# EPICS StreamDevice protocol: pt2025Sup/pt2025.proto
terminator = CR LF;

# catch field strengths
getFieldAuto {
  in  "%s";
}
